FUNCTION F_StringToTarg
VAR_INPUT
   StringToConvert : T_MaxString;
END_VAR
VAR_IN_OUT
   Targ : T_ARG;
END_VAR
VAR
   b : POINTER TO BOOL;
   b8 : POINTER TO BYTE;
   w : POINTER TO WORD;
   dw : POINTER TO DWORD;
   usi : POINTER TO USINT;
   si : POINTER TO SINT;
   ui : POINTER TO UINT;
   i : POINTER TO INT;
   udi : POINTER TO UDINT;
   di : POINTER TO DINT;
   str : POINTER TO STRING;
   re : POINTER TO REAL;
   lr : POINTER TO LREAL;
END_VAR

CASE Targ.eType OF

   E_ArgType.ARGTYPE_BOOL:
      b := Targ.pData;
      b^ := TO_BOOL(StringToConvert);

   E_ArgType.ARGTYPE_BYTE:
      b8 := Targ.pData;
      b8^ := TO_BYTE(StringToConvert);

   E_ArgType.ARGTYPE_WORD:
      w := Targ.pData;
      w^ := TO_WORD(StringToConvert);

   E_ArgType.ARGTYPE_DWORD:
      dw := Targ.pData;
      dw^ := TO_DWORD(StringToConvert);

   E_ArgType.ARGTYPE_USINT:
      usi := Targ.pData;
      usi^ := TO_USINT(StringToConvert);

   E_ArgType.ARGTYPE_SINT:
      si := Targ.pData;
      si^ := TO_SINT(StringToConvert);

   E_ArgType.ARGTYPE_UINT:
      ui := Targ.pData;
      ui^ := TO_UINT(StringToConvert);

   E_ArgType.ARGTYPE_INT:
      i := Targ.pData;
      i^ := TO_INT(StringToConvert);

   E_ArgType.ARGTYPE_UDINT:
      udi := Targ.pData;
      udi^ := TO_UDINT(StringToConvert);

   E_ArgType.ARGTYPE_DINT:
      di := Targ.pData;
      di^ := TO_DINT(StringToConvert);

   E_ArgType.ARGTYPE_STRING:
      str := Targ.pData;
      str^ := TO_STRING(StringToConvert);

   E_ArgType.ARGTYPE_REAL:
      re := Targ.pData;
      re^ := TO_REAL(StringToConvert);

   E_ArgType.ARGTYPE_LREAL:
      lr := Targ.pData;
      lr^ := TO_LREAL(StringToConvert);

ELSE
   F_LogWarning(
      CONCAT(
         'Unsupported type in Targ for string conversion: ',
         TO_STRING(Targ.eType)
      )
   );
END_CASE

END_FUNCTION

(* stored: Version 1.1.0.1, ProductVersion 3.1.4026.12
   POU F_StringToTarg: Id {cb329947-cdb8-0d3d-0d78-bac48c20f1a6}, SpecialFunc None *)
